FUNCTION_BLOCK INTIME (* Composite Function Block Type *)
  (* Standard: 61499-2 *)
  (* Version 0.0, 09/08/2022, Pranay Jhunjhunwala, UoA, template *)
  PACKAGE Main;
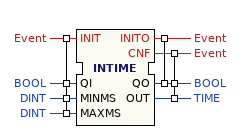
  EVENT_INPUT
    INIT WITH QI, MINMS, MAXMS; (* Initialization Request *)
  END_EVENT
  EVENT_OUTPUT
    INITO WITH QO; (* Initialization Confirm *)
    CNF WITH QO, OUT; (* Execution Confirmation *)
  END_EVENT
  VAR_INPUT
    QI : BOOL; (* Input event qualifier *)
    MINMS : DINT;
    MAXMS : DINT;
  END_VAR
  VAR_OUTPUT
    QO : BOOL; (* Output event qualifier *)
    OUT : TIME;
  END_VAR
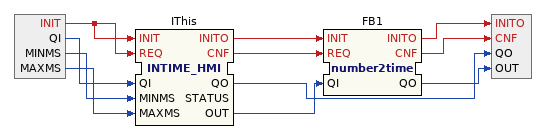
  FBS
    FB1 : number2time;
    IThis : INTIME_HMI;
  END_FBS
  EVENT_CONNECTIONS
    FB1.INITO TO INITO;
    FB1.CNF TO CNF;
    INIT TO IThis.INIT;
    IThis.INITO TO FB1.INIT;
    IThis.CNF TO FB1.REQ;
    INIT TO IThis.REQ;
  END_CONNECTIONS
  DATA_CONNECTIONS
    FB1.QO TO OUT;
    QI TO IThis.QI;
    MINMS TO IThis.MINMS;
    MAXMS TO IThis.MAXMS;
    IThis.QO TO QO;
    IThis.OUT TO FB1.QI;
  END_CONNECTIONS
END_FUNCTION_BLOCK
